// TIA Portal V17 export
// export: Created 2024-09-02T12:50:16.9080153Z, ExportSetting WithDefaults, DisplayName Totally Integrated Automation Portal, DisplayVersion V17, DisplayName TIA Portal Openness, DisplayVersion V17, DisplayName TIA Portal Version Control Interface, DisplayVersion V17, DisplayName STEP 7 Professional, DisplayVersion V17, DisplayName STEP 7 Safety, DisplayVersion V17, DisplayName WinCC Professional, DisplayVersion V17
DATA_BLOCK "AnwDB_StructureSelection_OP70"   // DB256
{ S7_Optimized_Access := 'TRUE'; DB_Accessible_From_OPC_UA := 'FALSE' }
AUTHOR : OlegFuehrus
FAMILY : BA
NAME : BA
VERSION : 0.1
// stored: AutoNumber false, DBAccessibleFromOPCUA false, IsOnlyStoredInLoadMemory false, IsRetainMemResEnabled true, IsWriteProtectedInAS false, MemoryReserve 60, RetainMemoryReserve 60
   VAR RETAIN
      Unit { ExternalWritable := 'False'} : Struct
         Camera { ExternalWritable := 'False'} : Bool;
         Gripper { ExternalWritable := 'False'} : Bool;
         Screwdriver { ExternalWritable := 'False'} : Bool;
         Deactiv_Res4 { ExternalWritable := 'False'} : Bool;
         Deactiv_Res5 { ExternalWritable := 'False'} : Bool;
         Deactiv_Res6 { ExternalWritable := 'False'} : Bool;
      END_STRUCT;
      NutRunner { ExternalWritable := 'False'} : Struct
         Deactiv_GR1 { ExternalWritable := 'False'} : Array[1..32] of Bool;
         Deactiv_GR2 { ExternalWritable := 'False'} : Array[1..32] of Bool;
      END_STRUCT;
      NutRunnerGroup { ExternalWritable := 'False'} : Struct
         Deactiv_Gruppe { ExternalWritable := 'False'} : Array[1..8] of Bool;
      END_STRUCT;
      CycleType { ExternalWritable := 'False'} : Struct
         Singel_Step { ExternalWritable := 'False'} : Bool;
         Service { ExternalWritable := 'False'} : Bool;
         MES_OFF { ExternalWritable := 'False'} : Bool;
         Bypass_DamperCaps_FEED { ExternalWritable := 'False'} : Bool;
         fpBypass_DamperCaps_FEED { ExternalWritable := 'False'} : Bool;
         fnBypass_DamperCaps_FEED { ExternalWritable := 'False'} : Bool;
         Bypass_DamperCaps_CAM { ExternalWritable := 'False'} : Bool;
         fpBypass_DamperCaps_CAM { ExternalWritable := 'False'} : Bool;
         fnBypass_DamperCaps_CAM { ExternalWritable := 'False'} : Bool;
      END_STRUCT;
      UserDefine { ExternalWritable := 'False'} : Struct
         IbmMode { ExternalWritable := 'False'} : Bool;
         Deactiv_Res3 { ExternalWritable := 'False'} : Bool;
         Deactiv_Res4 { ExternalWritable := 'False'} : Bool;
         Deactiv_Res5 { ExternalWritable := 'False'} : Bool;
         Deactiv_Res6 { ExternalWritable := 'False'} : Bool;
         Deactiv_Res7 { ExternalWritable := 'False'} : Bool;
      END_STRUCT;
   END_VAR
BEGIN
END_DATA_BLOCK
